// TwinCAT 3 PLC project IO_External_Task
// ProgramVersion: 3.1.4026.19
// libraries:
//   Tc2_Standard, * (Beckhoff Automation GmbH)
//   Tc2_System, * (Beckhoff Automation GmbH)
//   Tc3_Module, * (Beckhoff Automation GmbH)
// project tree:
//   DUTs/EtherCAT模組/ DI570.TcDUT, DO570.TcDUT
//   DUTs/ In_16_To_PLC.TcDUT, Out_16_To_PLC.TcDUT
//   GVLs/ EtherCAT.TcGVL, MainIO.TcGVL
//   / Main_IO_Task.TcTTO
//   POUs/IO轉換/ AI_force.TcPOU, IO_force.TcPOU
//   POUs/IO轉換/控制櫃/ Mod101.TcPOU, Mod102.TcPOU, Mod103.TcPOU, Mod104.TcPOU, Mod105.TcPOU, Mod106.TcPOU, Mod107.TcPOU
//   POUs/ MAIN.TcPOU
// (motion and I/O tree: see PLC project main)
// real-time tasks:
//   TASK Main_IO_Task: cycle T#2ms, priority 6, ADS port 353
//   TASK PlcTask: cycle T#10ms, priority 14, ADS port 350
//   TASK Conveyor: cycle T#10ms, priority 22, ADS port 355
// variable links:
//   External_Conveyor_system Instance <-> IO_External_Task/IO_External_Task Instance
//     PlcTask Inputs/IO.i101 <-> Main_IO_Task Outputs/MainIO.IO101.In[1]
//     PlcTask Inputs/IO.i102 <-> Main_IO_Task Outputs/MainIO.IO101.In[2]
//     PlcTask Inputs/IO.i103 <-> Main_IO_Task Outputs/MainIO.IO101.In[3]
//     PlcTask Inputs/IO.i104 <-> Main_IO_Task Outputs/MainIO.IO101.In[4]
//     PlcTask Inputs/IO.i105 <-> Main_IO_Task Outputs/MainIO.IO101.In[5]
//     PlcTask Inputs/IO.i106 <-> Main_IO_Task Outputs/MainIO.IO101.In[6]
//     PlcTask Inputs/IO.i107 <-> Main_IO_Task Outputs/MainIO.IO101.In[7]
//     PlcTask Inputs/IO.i108 <-> Main_IO_Task Outputs/MainIO.IO101.In[8]
//     PlcTask Inputs/IO.i109 <-> Main_IO_Task Outputs/MainIO.IO101.In[9]
//     PlcTask Inputs/IO.i110 <-> Main_IO_Task Outputs/MainIO.IO101.In[10]
//     PlcTask Inputs/IO.i111 <-> Main_IO_Task Outputs/MainIO.IO101.In[11]
//     PlcTask Inputs/IO.i112 <-> Main_IO_Task Outputs/MainIO.IO101.In[12]
//     PlcTask Inputs/IO.i113 <-> Main_IO_Task Outputs/MainIO.IO101.In[13]
//     PlcTask Inputs/IO.i114 <-> Main_IO_Task Outputs/MainIO.IO101.In[14]
//     PlcTask Inputs/IO.i115 <-> Main_IO_Task Outputs/MainIO.IO101.In[15]
//     PlcTask Inputs/IO.i116 <-> Main_IO_Task Outputs/MainIO.IO101.In[16]
//     PlcTask Inputs/IO.i201 <-> Main_IO_Task Outputs/MainIO.IO102.In[1]
//     PlcTask Inputs/IO.i202 <-> Main_IO_Task Outputs/MainIO.IO102.In[2]
//     PlcTask Inputs/IO.i203 <-> Main_IO_Task Outputs/MainIO.IO102.In[3]
//     PlcTask Inputs/IO.i204 <-> Main_IO_Task Outputs/MainIO.IO102.In[4]
//     PlcTask Inputs/IO.i205 <-> Main_IO_Task Outputs/MainIO.IO102.In[5]
//     PlcTask Inputs/IO.i206 <-> Main_IO_Task Outputs/MainIO.IO102.In[6]
//     PlcTask Inputs/IO.i207 <-> Main_IO_Task Outputs/MainIO.IO102.In[7]
//     PlcTask Inputs/IO.i208 <-> Main_IO_Task Outputs/MainIO.IO102.In[8]
//     PlcTask Inputs/IO.i209 <-> Main_IO_Task Outputs/MainIO.IO102.In[9]
//     PlcTask Inputs/IO.i210 <-> Main_IO_Task Outputs/MainIO.IO102.In[10]
//     PlcTask Inputs/IO.i211 <-> Main_IO_Task Outputs/MainIO.IO102.In[11]
//     PlcTask Inputs/IO.i212 <-> Main_IO_Task Outputs/MainIO.IO102.In[12]
//     PlcTask Inputs/IO.i213 <-> Main_IO_Task Outputs/MainIO.IO102.In[13]
//     PlcTask Inputs/IO.i214 <-> Main_IO_Task Outputs/MainIO.IO102.In[14]
//     PlcTask Inputs/IO.i215 <-> Main_IO_Task Outputs/MainIO.IO102.In[15]
//     PlcTask Inputs/IO.i216 <-> Main_IO_Task Outputs/MainIO.IO102.In[16]
//     PlcTask Inputs/IO.i301 <-> Main_IO_Task Outputs/MainIO.IO103.In[1]
//     PlcTask Inputs/IO.i302 <-> Main_IO_Task Outputs/MainIO.IO103.In[2]
//     PlcTask Inputs/IO.i303 <-> Main_IO_Task Outputs/MainIO.IO103.In[3]
//     PlcTask Inputs/IO.i304 <-> Main_IO_Task Outputs/MainIO.IO103.In[4]
//     PlcTask Inputs/IO.i305 <-> Main_IO_Task Outputs/MainIO.IO103.In[5]
//     PlcTask Inputs/IO.i306 <-> Main_IO_Task Outputs/MainIO.IO103.In[6]
//     PlcTask Inputs/IO.i307 <-> Main_IO_Task Outputs/MainIO.IO103.In[7]
//     PlcTask Inputs/IO.i308 <-> Main_IO_Task Outputs/MainIO.IO103.In[8]
//     PlcTask Inputs/IO.i309 <-> Main_IO_Task Outputs/MainIO.IO103.In[9]
//     PlcTask Inputs/IO.i310 <-> Main_IO_Task Outputs/MainIO.IO103.In[10]
//     PlcTask Inputs/IO.i311 <-> Main_IO_Task Outputs/MainIO.IO103.In[11]
//     PlcTask Inputs/IO.i312 <-> Main_IO_Task Outputs/MainIO.IO103.In[12]
//     PlcTask Inputs/IO.i313 <-> Main_IO_Task Outputs/MainIO.IO103.In[13]
//     PlcTask Inputs/IO.i314 <-> Main_IO_Task Outputs/MainIO.IO103.In[14]
//     PlcTask Inputs/IO.i315 <-> Main_IO_Task Outputs/MainIO.IO103.In[15]
//     PlcTask Inputs/IO.i316 <-> Main_IO_Task Outputs/MainIO.IO103.In[16]
//     PlcTask Inputs/IO.i401 <-> Main_IO_Task Outputs/MainIO.IO104.In[1]
//     PlcTask Inputs/IO.i402 <-> Main_IO_Task Outputs/MainIO.IO104.In[2]
//     PlcTask Inputs/IO.i403 <-> Main_IO_Task Outputs/MainIO.IO104.In[3]
//     PlcTask Inputs/IO.i404 <-> Main_IO_Task Outputs/MainIO.IO104.In[4]
//     PlcTask Inputs/IO.i405 <-> Main_IO_Task Outputs/MainIO.IO104.In[5]
//     PlcTask Inputs/IO.i406 <-> Main_IO_Task Outputs/MainIO.IO104.In[6]
//     PlcTask Inputs/IO.i407 <-> Main_IO_Task Outputs/MainIO.IO104.In[7]
//     PlcTask Inputs/IO.i408 <-> Main_IO_Task Outputs/MainIO.IO104.In[8]
//     PlcTask Inputs/IO.i409 <-> Main_IO_Task Outputs/MainIO.IO104.In[9]
//     PlcTask Inputs/IO.i410 <-> Main_IO_Task Outputs/MainIO.IO104.In[10]
//     PlcTask Inputs/IO.i411 <-> Main_IO_Task Outputs/MainIO.IO104.In[11]
//     PlcTask Inputs/IO.i412 <-> Main_IO_Task Outputs/MainIO.IO104.In[12]
//     PlcTask Inputs/IO.i413 <-> Main_IO_Task Outputs/MainIO.IO104.In[13]
//     PlcTask Inputs/IO.i414 <-> Main_IO_Task Outputs/MainIO.IO104.In[14]
//     PlcTask Inputs/IO.i415 <-> Main_IO_Task Outputs/MainIO.IO104.In[15]
//     PlcTask Inputs/IO.i416 <-> Main_IO_Task Outputs/MainIO.IO104.In[16]
//     PlcTask Outputs/IO.q101 <-> Main_IO_Task Inputs/MainIO.IO105.Out[1]
//     PlcTask Outputs/IO.q102 <-> Main_IO_Task Inputs/MainIO.IO105.Out[2]
//     PlcTask Outputs/IO.q103 <-> Main_IO_Task Inputs/MainIO.IO105.Out[3]
//     PlcTask Outputs/IO.q104 <-> Main_IO_Task Inputs/MainIO.IO105.Out[4]
//     PlcTask Outputs/IO.q105 <-> Main_IO_Task Inputs/MainIO.IO105.Out[5]
//     PlcTask Outputs/IO.q106 <-> Main_IO_Task Inputs/MainIO.IO105.Out[6]
//     PlcTask Outputs/IO.q107 <-> Main_IO_Task Inputs/MainIO.IO105.Out[7]
//     PlcTask Outputs/IO.q108 <-> Main_IO_Task Inputs/MainIO.IO105.Out[8]
//     PlcTask Outputs/IO.q109 <-> Main_IO_Task Inputs/MainIO.IO105.Out[9]
//     PlcTask Outputs/IO.q110 <-> Main_IO_Task Inputs/MainIO.IO105.Out[10]
//     PlcTask Outputs/IO.q111 <-> Main_IO_Task Inputs/MainIO.IO105.Out[11]
//     PlcTask Outputs/IO.q112 <-> Main_IO_Task Inputs/MainIO.IO105.Out[12]
//     PlcTask Outputs/IO.q113 <-> Main_IO_Task Inputs/MainIO.IO105.Out[13]
//     PlcTask Outputs/IO.q114 <-> Main_IO_Task Inputs/MainIO.IO105.Out[14]
//     PlcTask Outputs/IO.q115 <-> Main_IO_Task Inputs/MainIO.IO105.Out[15]
//     PlcTask Outputs/IO.q116 <-> Main_IO_Task Inputs/MainIO.IO105.Out[16]
//     PlcTask Outputs/IO.q201 <-> Main_IO_Task Inputs/MainIO.IO106.Out[1]
//     PlcTask Outputs/IO.q202 <-> Main_IO_Task Inputs/MainIO.IO106.Out[2]
//     PlcTask Outputs/IO.q203 <-> Main_IO_Task Inputs/MainIO.IO106.Out[3]
//     PlcTask Outputs/IO.q204 <-> Main_IO_Task Inputs/MainIO.IO106.Out[4]
//     PlcTask Outputs/IO.q205 <-> Main_IO_Task Inputs/MainIO.IO106.Out[5]
//     PlcTask Outputs/IO.q206 <-> Main_IO_Task Inputs/MainIO.IO106.Out[6]
//     PlcTask Outputs/IO.q207 <-> Main_IO_Task Inputs/MainIO.IO106.Out[7]
//     PlcTask Outputs/IO.q208 <-> Main_IO_Task Inputs/MainIO.IO106.Out[8]
//     PlcTask Outputs/IO.q209 <-> Main_IO_Task Inputs/MainIO.IO106.Out[9]
//     PlcTask Outputs/IO.q210 <-> Main_IO_Task Inputs/MainIO.IO106.Out[10]
//     PlcTask Outputs/IO.q211 <-> Main_IO_Task Inputs/MainIO.IO106.Out[11]
//     PlcTask Outputs/IO.q212 <-> Main_IO_Task Inputs/MainIO.IO106.Out[12]
//     PlcTask Outputs/IO.q213 <-> Main_IO_Task Inputs/MainIO.IO106.Out[13]
//     PlcTask Outputs/IO.q214 <-> Main_IO_Task Inputs/MainIO.IO106.Out[14]
//     PlcTask Outputs/IO.q215 <-> Main_IO_Task Inputs/MainIO.IO106.Out[15]
//     PlcTask Outputs/IO.q216 <-> Main_IO_Task Inputs/MainIO.IO106.Out[16]
//     PlcTask Outputs/IO.q301 <-> Main_IO_Task Inputs/MainIO.IO107.Out[1]
//     PlcTask Outputs/IO.q302 <-> Main_IO_Task Inputs/MainIO.IO107.Out[2]
//     PlcTask Outputs/IO.q303 <-> Main_IO_Task Inputs/MainIO.IO107.Out[3]
//     PlcTask Outputs/IO.q304 <-> Main_IO_Task Inputs/MainIO.IO107.Out[4]
//     PlcTask Outputs/IO.q305 <-> Main_IO_Task Inputs/MainIO.IO107.Out[5]
//     PlcTask Outputs/IO.q306 <-> Main_IO_Task Inputs/MainIO.IO107.Out[6]
//     PlcTask Outputs/IO.q307 <-> Main_IO_Task Inputs/MainIO.IO107.Out[7]
//     PlcTask Outputs/IO.q308 <-> Main_IO_Task Inputs/MainIO.IO107.Out[8]
//     PlcTask Outputs/IO.q309 <-> Main_IO_Task Inputs/MainIO.IO107.Out[9]
//     PlcTask Outputs/IO.q310 <-> Main_IO_Task Inputs/MainIO.IO107.Out[10]
//     PlcTask Outputs/IO.q311 <-> Main_IO_Task Inputs/MainIO.IO107.Out[11]
//     PlcTask Outputs/IO.q312 <-> Main_IO_Task Inputs/MainIO.IO107.Out[12]
//     PlcTask Outputs/IO.q313 <-> Main_IO_Task Inputs/MainIO.IO107.Out[13]
//     PlcTask Outputs/IO.q314 <-> Main_IO_Task Inputs/MainIO.IO107.Out[14]
//     PlcTask Outputs/IO.q315 <-> Main_IO_Task Inputs/MainIO.IO107.Out[15]
//     PlcTask Outputs/IO.q316 <-> Main_IO_Task Inputs/MainIO.IO107.Out[16]

CONFIGURATION IO_External_Task
    RESOURCE PLC ON TwinCAT3
        TASK Main_IO_Task(INTERVAL := T#2ms, PRIORITY := 6);
        PROGRAM MAIN WITH Main_IO_Task : MAIN;
    END_RESOURCE
END_CONFIGURATION

// ---- DUTs/EtherCAT模組/DI570.TcDUT
TYPE DI570 :
STRUCT
	ModType : STRING := 'KEBA DI570';
	Input AT %I*:ARRAY [1..18] OF BOOL;
	WcState AT %I*:BOOL;
	InputToggle AT %I*:BOOL;
	State AT %I*:UINT;
END_STRUCT
END_TYPE

// ---- DUTs/EtherCAT模組/DO570.TcDUT
TYPE DO570 :
STRUCT
	ModType : STRING := 'KEBA DO570';
	WcState AT %I*:BOOL;
	State AT %I*:UINT;
	Output_ShortCircuit AT %I*:ARRAY [1..16] OF BOOL;
	Output AT %Q*:ARRAY [1..16] OF BOOL;
END_STRUCT
END_TYPE

// ---- DUTs/In_16_To_PLC.TcDUT
TYPE In_16_To_PLC :
STRUCT
	In AT %Q*:ARRAY [1..16] OF BOOL;
END_STRUCT
END_TYPE

// ---- DUTs/Out_16_To_PLC.TcDUT
TYPE Out_16_To_PLC :
STRUCT
	Out AT %I*:ARRAY [1..16] OF BOOL;
END_STRUCT
END_TYPE

// ---- GVLs/EtherCAT.TcGVL
{attribute 'qualified_only'}
VAR_GLOBAL
	// 主控制櫃 控制器
	LoadMod_1 :DI570;
	LoadMod_2 :DI570;
	LoadMod_3 :DI570;
	LoadMod_4 :DI570;
	
	LoadMod_5 :DO570;
	LoadMod_6 :DO570;
	LoadMod_7 :DO570;
END_VAR

// ---- GVLs/MainIO.TcGVL
{attribute 'qualified_onlY0'}
VAR_GLOBAL
	//
	IO101: In_16_To_PLC;
	//
	IO102: In_16_To_PLC;
	//
	IO103: In_16_To_PLC;
	//
	IO104: In_16_To_PLC;
	
	
	//
	IO105: Out_16_To_PLC;
	//
	IO106: Out_16_To_PLC;
	//
	IO107: Out_16_To_PLC;
	
	
	

	IO101_s : WORD;
	IO102_s : WORD;
	IO103_s : WORD;
	IO104_s : WORD;
	IO105_s : WORD;
	IO106_s : WORD;
	IO107_s : WORD;
	
	IO101_f : WORD;
	IO102_f : WORD;
	IO103_f : WORD;
	IO104_f : WORD;
	IO105_f : WORD;
	IO106_f : WORD;
	IO107_f : WORD;
END_VAR

// ---- POUs/MAIN.TcPOU
PROGRAM MAIN
VAR
END_VAR

Mod101();
Mod102();
Mod103();
Mod104();
Mod105();
Mod106();
Mod107();

END_PROGRAM

// ---- POUs/IO轉換/控制櫃/Mod101.TcPOU
PROGRAM Mod101
VAR
	IO_f : ARRAY [1..16] OF IO_force;
	
	i: SINT;
END_VAR

	// 輸入模組1
	FOR i := 1 TO 16 DO
		IO_f[i](Raw_IO := EtherCAT.LoadMod_1.Input[i], Out =>MainIO.IO101.In[i]);
	END_FOR
	
	
	MainIO.IO101_s.0 := IO_f[1].Out;
	MainIO.IO101_s.1 := IO_f[2].Out;
	MainIO.IO101_s.2 := IO_f[3].Out;
	MainIO.IO101_s.3 := IO_f[4].Out;
	MainIO.IO101_s.4 := IO_f[5].Out;
	MainIO.IO101_s.5 := IO_f[6].Out;
	MainIO.IO101_s.6 := IO_f[7].Out;
	MainIO.IO101_s.7 := IO_f[8].Out;
	MainIO.IO101_s.8 := IO_f[9].Out;
	MainIO.IO101_s.9 := IO_f[10].Out;
	MainIO.IO101_s.10 := IO_f[11].Out;
	MainIO.IO101_s.11 := IO_f[12].Out;
	MainIO.IO101_s.12 := IO_f[13].Out;
	MainIO.IO101_s.13 := IO_f[14].Out;
	MainIO.IO101_s.14 := IO_f[15].Out;
	MainIO.IO101_s.15 := IO_f[16].Out;
	
	MainIO.io101_f.0 := IO_f[1].ForceEnable;
	MainIO.io101_f.1 := IO_f[2].ForceEnable;
	MainIO.io101_f.2 := IO_f[3].ForceEnable;
	MainIO.io101_f.3 := IO_f[4].ForceEnable;
	MainIO.io101_f.4 := IO_f[5].ForceEnable;
	MainIO.io101_f.5 := IO_f[6].ForceEnable;
	MainIO.io101_f.6 := IO_f[7].ForceEnable;
	MainIO.io101_f.7 := IO_f[8].ForceEnable;
	MainIO.io101_f.8 := IO_f[9].ForceEnable;
	MainIO.io101_f.9 := IO_f[10].ForceEnable;
	MainIO.io101_f.10 := IO_f[11].ForceEnable;
	MainIO.io101_f.11 := IO_f[12].ForceEnable;
	MainIO.io101_f.12 := IO_f[13].ForceEnable;
	MainIO.io101_f.13 := IO_f[14].ForceEnable;
	MainIO.io101_f.14 := IO_f[15].ForceEnable;
	MainIO.io101_f.15 := IO_f[16].ForceEnable;

END_PROGRAM

// ---- POUs/IO轉換/IO_force.TcPOU
FUNCTION_BLOCK IO_force
VAR_INPUT
	Raw_IO : BOOL;
END_VAR

VAR_OUTPUT
	Out : BOOL;
END_VAR

VAR
	ForceEnable : BOOL;
	ForceStatus : BOOL;
END_VAR

IF NOT ForceEnable THEN
	OUT := Raw_IO;
ELSE
	OUT := ForceStatus;
END_IF

END_FUNCTION_BLOCK

// ---- POUs/IO轉換/控制櫃/Mod102.TcPOU
PROGRAM Mod102
VAR
	IO_f : ARRAY [1..16] OF IO_force;
	i: SINT;
END_VAR

	// 輸入模組1
	FOR i := 1 TO 16 DO
		IO_f[i](Raw_IO := EtherCAT.LoadMod_2.Input[i], Out =>MainIO.io102.In[i]);
	END_FOR
	
	
	MainIO.io102_s.0 := IO_f[1].Out;
	MainIO.io102_s.1 := IO_f[2].Out;
	MainIO.io102_s.2 := IO_f[3].Out;
	MainIO.io102_s.3 := IO_f[4].Out;
	MainIO.io102_s.4 := IO_f[5].Out;
	MainIO.io102_s.5 := IO_f[6].Out;
	MainIO.io102_s.6 := IO_f[7].Out;
	MainIO.io102_s.7 := IO_f[8].Out;
	MainIO.io102_s.8 := IO_f[9].Out;
	MainIO.io102_s.9 := IO_f[10].Out;
	MainIO.io102_s.10 := IO_f[11].Out;
	MainIO.io102_s.11 := IO_f[12].Out;
	MainIO.io102_s.12 := IO_f[13].Out;
	MainIO.io102_s.13 := IO_f[14].Out;
	MainIO.io102_s.14 := IO_f[15].Out;
	MainIO.io102_s.15 := IO_f[16].Out;
	
	MainIO.io102_f.0 := IO_f[1].ForceEnable;
	MainIO.io102_f.1 := IO_f[2].ForceEnable;
	MainIO.io102_f.2 := IO_f[3].ForceEnable;
	MainIO.io102_f.3 := IO_f[4].ForceEnable;
	MainIO.io102_f.4 := IO_f[5].ForceEnable;
	MainIO.io102_f.5 := IO_f[6].ForceEnable;
	MainIO.io102_f.6 := IO_f[7].ForceEnable;
	MainIO.io102_f.7 := IO_f[8].ForceEnable;
	MainIO.io102_f.8 := IO_f[9].ForceEnable;
	MainIO.io102_f.9 := IO_f[10].ForceEnable;
	MainIO.io102_f.10 := IO_f[11].ForceEnable;
	MainIO.io102_f.11 := IO_f[12].ForceEnable;
	MainIO.io102_f.12 := IO_f[13].ForceEnable;
	MainIO.io102_f.13 := IO_f[14].ForceEnable;
	MainIO.io102_f.14 := IO_f[15].ForceEnable;
	MainIO.io102_f.15 := IO_f[16].ForceEnable;

END_PROGRAM

// ---- POUs/IO轉換/控制櫃/Mod103.TcPOU
PROGRAM Mod103
VAR
	IO_f : ARRAY [1..16] OF IO_force;
	i: SINT;
END_VAR

	// 輸入模組1
	FOR i := 1 TO 16 DO
		IO_f[i](Raw_IO := EtherCAT.LoadMod_3.Input[i], Out =>MainIO.io103.In[i]);
	END_FOR
	
	
	MainIO.io103_s.0 := IO_f[1].Out;
	MainIO.io103_s.1 := IO_f[2].Out;
	MainIO.io103_s.2 := IO_f[3].Out;
	MainIO.io103_s.3 := IO_f[4].Out;
	MainIO.io103_s.4 := IO_f[5].Out;
	MainIO.io103_s.5 := IO_f[6].Out;
	MainIO.io103_s.6 := IO_f[7].Out;
	MainIO.io103_s.7 := IO_f[8].Out;
	MainIO.io103_s.8 := IO_f[9].Out;
	MainIO.io103_s.9 := IO_f[10].Out;
	MainIO.io103_s.10 := IO_f[11].Out;
	MainIO.io103_s.11 := IO_f[12].Out;
	MainIO.io103_s.12 := IO_f[13].Out;
	MainIO.io103_s.13 := IO_f[14].Out;
	MainIO.io103_s.14 := IO_f[15].Out;
	MainIO.io103_s.15 := IO_f[16].Out;
	
	MainIO.io103_f.0 := IO_f[1].ForceEnable;
	MainIO.io103_f.1 := IO_f[2].ForceEnable;
	MainIO.io103_f.2 := IO_f[3].ForceEnable;
	MainIO.io103_f.3 := IO_f[4].ForceEnable;
	MainIO.io103_f.4 := IO_f[5].ForceEnable;
	MainIO.io103_f.5 := IO_f[6].ForceEnable;
	MainIO.io103_f.6 := IO_f[7].ForceEnable;
	MainIO.io103_f.7 := IO_f[8].ForceEnable;
	MainIO.io103_f.8 := IO_f[9].ForceEnable;
	MainIO.io103_f.9 := IO_f[10].ForceEnable;
	MainIO.io103_f.10 := IO_f[11].ForceEnable;
	MainIO.io103_f.11 := IO_f[12].ForceEnable;
	MainIO.io103_f.12 := IO_f[13].ForceEnable;
	MainIO.io103_f.13 := IO_f[14].ForceEnable;
	MainIO.io103_f.14 := IO_f[15].ForceEnable;
	MainIO.io103_f.15 := IO_f[16].ForceEnable;

END_PROGRAM

// ---- POUs/IO轉換/控制櫃/Mod104.TcPOU
PROGRAM Mod104
VAR
	IO_f : ARRAY [1..16] OF IO_force;
	i: SINT;
END_VAR

	// 輸入模組1
	FOR i := 1 TO 16 DO
		IO_f[i](Raw_IO := EtherCAT.LoadMod_4.Input[i], Out =>MainIO.io104.In[i]);
	END_FOR
	
	
	MainIO.io104_s.0 := IO_f[1].Out;
	MainIO.io104_s.1 := IO_f[2].Out;
	MainIO.io104_s.2 := IO_f[3].Out;
	MainIO.io104_s.3 := IO_f[4].Out;
	MainIO.io104_s.4 := IO_f[5].Out;
	MainIO.io104_s.5 := IO_f[6].Out;
	MainIO.io104_s.6 := IO_f[7].Out;
	MainIO.io104_s.7 := IO_f[8].Out;
	MainIO.io104_s.8 := IO_f[9].Out;
	MainIO.io104_s.9 := IO_f[10].Out;
	MainIO.io104_s.10 := IO_f[11].Out;
	MainIO.io104_s.11 := IO_f[12].Out;
	MainIO.io104_s.12 := IO_f[13].Out;
	MainIO.io104_s.13 := IO_f[14].Out;
	MainIO.io104_s.14 := IO_f[15].Out;
	MainIO.io104_s.15 := IO_f[16].Out;
	
	MainIO.io104_f.0 := IO_f[1].ForceEnable;
	MainIO.io104_f.1 := IO_f[2].ForceEnable;
	MainIO.io104_f.2 := IO_f[3].ForceEnable;
	MainIO.io104_f.3 := IO_f[4].ForceEnable;
	MainIO.io104_f.4 := IO_f[5].ForceEnable;
	MainIO.io104_f.5 := IO_f[6].ForceEnable;
	MainIO.io104_f.6 := IO_f[7].ForceEnable;
	MainIO.io104_f.7 := IO_f[8].ForceEnable;
	MainIO.io104_f.8 := IO_f[9].ForceEnable;
	MainIO.io104_f.9 := IO_f[10].ForceEnable;
	MainIO.io104_f.10 := IO_f[11].ForceEnable;
	MainIO.io104_f.11 := IO_f[12].ForceEnable;
	MainIO.io104_f.12 := IO_f[13].ForceEnable;
	MainIO.io104_f.13 := IO_f[14].ForceEnable;
	MainIO.io104_f.14 := IO_f[15].ForceEnable;
	MainIO.io104_f.15 := IO_f[16].ForceEnable;

END_PROGRAM

// ---- POUs/IO轉換/控制櫃/Mod105.TcPOU
PROGRAM Mod105
VAR
	IO_f : ARRAY [1..16] OF IO_force;
	
	i: SINT;
END_VAR

	// 輸入模組1
	FOR i := 1 TO 16 DO
		IO_f[i](Raw_IO := MainIO.IO105.Out[i], Out => EtherCAT.LoadMod_5.Output[i]);
	END_FOR
	
	
	MainIO.IO105_s.0 := IO_f[1].Out;
	MainIO.IO105_s.1 := IO_f[2].Out;
	MainIO.IO105_s.2 := IO_f[3].Out;
	MainIO.IO105_s.3 := IO_f[4].Out;
	MainIO.IO105_s.4 := IO_f[5].Out;
	MainIO.IO105_s.5 := IO_f[6].Out;
	MainIO.IO105_s.6 := IO_f[7].Out;
	MainIO.IO105_s.7 := IO_f[8].Out;
	MainIO.IO105_s.8 := IO_f[9].Out;
	MainIO.IO105_s.9 := IO_f[10].Out;
	MainIO.IO105_s.10 := IO_f[11].Out;
	MainIO.IO105_s.11 := IO_f[12].Out;
	MainIO.IO105_s.12 := IO_f[13].Out;
	MainIO.IO105_s.13 := IO_f[14].Out;
	MainIO.IO105_s.14 := IO_f[15].Out;
	MainIO.IO105_s.15 := IO_f[16].Out;
	
	MainIO.IO105_f.0 := IO_f[1].ForceEnable;
	MainIO.IO105_f.1 := IO_f[2].ForceEnable;
	MainIO.IO105_f.2 := IO_f[3].ForceEnable;
	MainIO.IO105_f.3 := IO_f[4].ForceEnable;
	MainIO.IO105_f.4 := IO_f[5].ForceEnable;
	MainIO.IO105_f.5 := IO_f[6].ForceEnable;
	MainIO.IO105_f.6 := IO_f[7].ForceEnable;
	MainIO.IO105_f.7 := IO_f[8].ForceEnable;
	MainIO.IO105_f.8 := IO_f[9].ForceEnable;
	MainIO.IO105_f.9 := IO_f[10].ForceEnable;
	MainIO.IO105_f.10 := IO_f[11].ForceEnable;
	MainIO.IO105_f.11 := IO_f[12].ForceEnable;
	MainIO.IO105_f.12 := IO_f[13].ForceEnable;
	MainIO.IO105_f.13 := IO_f[14].ForceEnable;
	MainIO.IO105_f.14 := IO_f[15].ForceEnable;
	MainIO.IO105_f.15 := IO_f[16].ForceEnable;

END_PROGRAM

// ---- POUs/IO轉換/控制櫃/Mod106.TcPOU
PROGRAM Mod106
VAR
	IO_f : ARRAY [1..16] OF IO_force;
	
	i: SINT;
END_VAR

	// 輸入模組1
	FOR i := 1 TO 16 DO
		IO_f[i](Raw_IO := MainIO.IO106.Out[i], Out => EtherCAT.LoadMod_6.Output[i]);
	END_FOR
	
	
	MainIO.IO106_s.0 := IO_f[1].Out;
	MainIO.IO106_s.1 := IO_f[2].Out;
	MainIO.IO106_s.2 := IO_f[3].Out;
	MainIO.IO106_s.3 := IO_f[4].Out;
	MainIO.IO106_s.4 := IO_f[5].Out;
	MainIO.IO106_s.5 := IO_f[6].Out;
	MainIO.IO106_s.6 := IO_f[7].Out;
	MainIO.IO106_s.7 := IO_f[8].Out;
	MainIO.IO106_s.8 := IO_f[9].Out;
	MainIO.IO106_s.9 := IO_f[10].Out;
	MainIO.IO106_s.10 := IO_f[11].Out;
	MainIO.IO106_s.11 := IO_f[12].Out;
	MainIO.IO106_s.12 := IO_f[13].Out;
	MainIO.IO106_s.13 := IO_f[14].Out;
	MainIO.IO106_s.14 := IO_f[15].Out;
	MainIO.IO106_s.15 := IO_f[16].Out;
	
	MainIO.IO106_f.0 := IO_f[1].ForceEnable;
	MainIO.IO106_f.1 := IO_f[2].ForceEnable;
	MainIO.IO106_f.2 := IO_f[3].ForceEnable;
	MainIO.IO106_f.3 := IO_f[4].ForceEnable;
	MainIO.IO106_f.4 := IO_f[5].ForceEnable;
	MainIO.IO106_f.5 := IO_f[6].ForceEnable;
	MainIO.IO106_f.6 := IO_f[7].ForceEnable;
	MainIO.IO106_f.7 := IO_f[8].ForceEnable;
	MainIO.IO106_f.8 := IO_f[9].ForceEnable;
	MainIO.IO106_f.9 := IO_f[10].ForceEnable;
	MainIO.IO106_f.10 := IO_f[11].ForceEnable;
	MainIO.IO106_f.11 := IO_f[12].ForceEnable;
	MainIO.IO106_f.12 := IO_f[13].ForceEnable;
	MainIO.IO106_f.13 := IO_f[14].ForceEnable;
	MainIO.IO106_f.14 := IO_f[15].ForceEnable;
	MainIO.IO106_f.15 := IO_f[16].ForceEnable;

END_PROGRAM

// ---- POUs/IO轉換/控制櫃/Mod107.TcPOU
PROGRAM Mod107
VAR
	IO_f : ARRAY [1..16] OF IO_force;
	
	i: SINT;
END_VAR

	// 輸入模組1
	FOR i := 1 TO 16 DO
		IO_f[i](Raw_IO := MainIO.IO107.Out[i], Out => EtherCAT.LoadMod_7.Output[i]);
	END_FOR
	
	
	MainIO.IO107_s.0 := IO_f[1].Out;
	MainIO.IO107_s.1 := IO_f[2].Out;
	MainIO.IO107_s.2 := IO_f[3].Out;
	MainIO.IO107_s.3 := IO_f[4].Out;
	MainIO.IO107_s.4 := IO_f[5].Out;
	MainIO.IO107_s.5 := IO_f[6].Out;
	MainIO.IO107_s.6 := IO_f[7].Out;
	MainIO.IO107_s.7 := IO_f[8].Out;
	MainIO.IO107_s.8 := IO_f[9].Out;
	MainIO.IO107_s.9 := IO_f[10].Out;
	MainIO.IO107_s.10 := IO_f[11].Out;
	MainIO.IO107_s.11 := IO_f[12].Out;
	MainIO.IO107_s.12 := IO_f[13].Out;
	MainIO.IO107_s.13 := IO_f[14].Out;
	MainIO.IO107_s.14 := IO_f[15].Out;
	MainIO.IO107_s.15 := IO_f[16].Out;
	
	MainIO.IO107_f.0 := IO_f[1].ForceEnable;
	MainIO.IO107_f.1 := IO_f[2].ForceEnable;
	MainIO.IO107_f.2 := IO_f[3].ForceEnable;
	MainIO.IO107_f.3 := IO_f[4].ForceEnable;
	MainIO.IO107_f.4 := IO_f[5].ForceEnable;
	MainIO.IO107_f.5 := IO_f[6].ForceEnable;
	MainIO.IO107_f.6 := IO_f[7].ForceEnable;
	MainIO.IO107_f.7 := IO_f[8].ForceEnable;
	MainIO.IO107_f.8 := IO_f[9].ForceEnable;
	MainIO.IO107_f.9 := IO_f[10].ForceEnable;
	MainIO.IO107_f.10 := IO_f[11].ForceEnable;
	MainIO.IO107_f.11 := IO_f[12].ForceEnable;
	MainIO.IO107_f.12 := IO_f[13].ForceEnable;
	MainIO.IO107_f.13 := IO_f[14].ForceEnable;
	MainIO.IO107_f.14 := IO_f[15].ForceEnable;
	MainIO.IO107_f.15 := IO_f[16].ForceEnable;

END_PROGRAM

// ---- POUs/IO轉換/AI_force.TcPOU
FUNCTION_BLOCK AI_force
VAR_INPUT
	Raw_IO : INT;
END_VAR

VAR_OUTPUT
	Out : INT;
END_VAR

VAR
	ForceEnable : BOOL;
	ForceValue : INT;
END_VAR

IF NOT ForceEnable THEN
	OUT := Raw_IO;
ELSE
	OUT := ForceValue;
END_IF

END_FUNCTION_BLOCK
